ABB RobotStudio station: Machina Testbed.rsstn

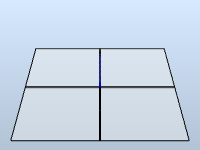
Station Machina Testbed (saved by RobotStudio 6.4.7120.133)
Controller IRB_4600_45kg_2.05m
  mechanical unit ROB_1: IRB4600_45_205_C_01, 6 joints, base frame (0, 0, 0) mm
Layout (positions relative to the parent item):
  - IRB4600_45_205_C_01 [mechanism, from Robots\IRB4600_45_205_C_G_01.rslib] at (0, 0, 0) mm; joint values [0, 0, 0, 0, 0.5236, 0] (rad or m)
